{attribute 'qualified_only'}
VAR_GLOBAL
	var01		:	INT;
END_VAR

(* stored: Version 1.1.0.1, ProductVersion 3.1.4020.6
   GVL GVL02: Id {72ec2962-9525-4b54-bffc-2e335e175d33} *)
